{attribute 'qualified_only'}
VAR_GLOBAL
		EtherCAT_Master_KLxxxx : EtherCAT_Master_KLxxxx_4053F38C;
		EtherCAT_Master_KLxxxx_1 : EtherCAT_Master_KLxxxx_1_8A657514;
		EtherCAT_Master_KLxxxx_2 : EtherCAT_Master_KLxxxx_2_B156B97E;
END_VAR

(* stored: Version 1.2.0.0, ProductVersion 3.1.4024.9
   GVL GVL_iXlinker: Id {201bad71-7910-4fb0-934c-11091a1718ed} *)
